// TIA Portal V15.1 export
// export: Created 2024-06-21T08:41:05.8674969Z, ExportSetting WithDefaults, DisplayName Totally Integrated Automation Portal, DisplayVersion V15.1 Update 5, DisplayName TIA Portal Openness, DisplayVersion V15.1 Update 5, DisplayName SINAMICS Startdrive Advanced, DisplayVersion V15.1, DisplayName G130, G150, S120, S150, SINAMICS MV, S210, DisplayVersion V15.1, DisplayName G110M, G120, G120C, G120D, G120P, DisplayVersion V15.1, DisplayName STEP 7 Professional, DisplayVersion V15.1 Update 5, DisplayName STEP 7 Safety, DisplayVersion V15.1, DisplayName WinCC Professional, DisplayVersion V15.1 Update 5, DisplayName SIMATIC Visualization Architect, DisplayVersion V15.1
FUNCTION_BLOCK "LGBDanfoss-FC302PN"   // FB6600, FBD
TITLE = LGBDanfoss-FC302PN
{ S7_Optimized_Access := 'TRUE' }
AUTHOR : VCC
FAMILY : Actuator
NAME : Danfoss
VERSION : 0.1
// ============================================================================  Block to control a frequency controller Danfoss FC302 on ProfiNET.  ============================================================================
// stored: AutoNumber false, IsIECCheckEnabled false, IsRetainMemResEnabled false, MemoryReserve 100, SetENOAutomatically False, UDAEnableTagReadback false
   VAR_INPUT
      I_ReferenceValueLSB { ExternalAccessible := 'False'; ExternalVisible := 'False'; ExternalWritable := 'False'} : Bool;   // Bit 0
      I_ReferenceValueMSB { ExternalAccessible := 'False'; ExternalVisible := 'False'; ExternalWritable := 'False'} : Bool;   // Bit 1
      I_DCBrake { ExternalAccessible := 'False'; ExternalVisible := 'False'; ExternalWritable := 'False'} : Bool;   // Bit 2
      I_Coasting { ExternalAccessible := 'False'; ExternalVisible := 'False'; ExternalWritable := 'False'} : Bool;   // Bit 3
      I_QuickStop { ExternalAccessible := 'False'; ExternalVisible := 'False'; ExternalWritable := 'False'} : Bool;   // Bit 4
      I_HoldOutputFreq { ExternalAccessible := 'False'; ExternalVisible := 'False'; ExternalWritable := 'False'} : Bool;   // Bit 5
      I_RampStopStart { ExternalAccessible := 'False'; ExternalVisible := 'False'; ExternalWritable := 'False'} : Bool;   // Bit 6
      I_Reset { ExternalAccessible := 'False'; ExternalVisible := 'False'; ExternalWritable := 'False'} : Bool;   // Bit 7
      I_Jog { ExternalAccessible := 'False'; ExternalVisible := 'False'; ExternalWritable := 'False'} : Bool;   // Bit 8
      I_RampSelection { ExternalAccessible := 'False'; ExternalVisible := 'False'; ExternalWritable := 'False'} : Bool;   // Bit 9
      I_DataValid { ExternalAccessible := 'False'; ExternalVisible := 'False'; ExternalWritable := 'False'} : Bool;   // Bit 10
      I_Relay01 { ExternalAccessible := 'False'; ExternalVisible := 'False'; ExternalWritable := 'False'} : Bool;   // Bit 11
      I_Relay04 { ExternalAccessible := 'False'; ExternalVisible := 'False'; ExternalWritable := 'False'} : Bool;   // Bit 12
      I_SetupSelectionLSB { ExternalAccessible := 'False'; ExternalVisible := 'False'; ExternalWritable := 'False'} : Bool;   // Bit 13
      I_SetupSelectionMSB { ExternalAccessible := 'False'; ExternalVisible := 'False'; ExternalWritable := 'False'} : Bool;   // Bit 14
      I_Reverse { ExternalAccessible := 'False'; ExternalVisible := 'False'; ExternalWritable := 'False'} : Bool;   // Bit 15
      C_HWSubInput { ExternalAccessible := 'False'; ExternalVisible := 'False'; ExternalWritable := 'False'} : HW_SUBMODULE;   // I/O
      C_HWSubOutput { ExternalAccessible := 'False'; ExternalVisible := 'False'; ExternalWritable := 'False'} : HW_SUBMODULE;   // I/O
      I_MRV_FC { ExternalAccessible := 'False'; ExternalVisible := 'False'; ExternalWritable := 'False'} : Real;   // Main Reference Value (0-4000Hex = 0 - 100 %)
      I_PCDIndex3 { ExternalAccessible := 'False'; ExternalVisible := 'False'; ExternalWritable := 'False'} : Int;   // Process data index 3
      I_PCDIndex4 { ExternalAccessible := 'False'; ExternalVisible := 'False'; ExternalWritable := 'False'} : Int;   // Process data index 4
      I_PCDIndex5 { ExternalAccessible := 'False'; ExternalVisible := 'False'; ExternalWritable := 'False'} : Int;   // Process data index 5
      I_PCDIndex6 { ExternalAccessible := 'False'; ExternalVisible := 'False'; ExternalWritable := 'False'} : Int;   // Process data index 6
      I_PCDIndex7 { ExternalAccessible := 'False'; ExternalVisible := 'False'; ExternalWritable := 'False'} : Int;   // Process data index 7
      I_PCDIndex8 { ExternalAccessible := 'False'; ExternalVisible := 'False'; ExternalWritable := 'False'} : Int;   // Process data index 8
      I_PCDIndex9 { ExternalAccessible := 'False'; ExternalVisible := 'False'; ExternalWritable := 'False'} : Int;   // Process data index 9
      I_PCDIndex10 { ExternalAccessible := 'False'; ExternalVisible := 'False'; ExternalWritable := 'False'} : Int;   // Process data index 10
   END_VAR
   VAR_OUTPUT
      O_FCReady { ExternalAccessible := 'False'; ExternalVisible := 'False'; ExternalWritable := 'False'} : Bool;
      O_DriveReady { ExternalAccessible := 'False'; ExternalVisible := 'False'; ExternalWritable := 'False'} : Bool;
      O_CoastingReady { ExternalAccessible := 'False'; ExternalVisible := 'False'; ExternalWritable := 'False'} : Bool;
      O_Trip { ExternalAccessible := 'False'; ExternalVisible := 'False'; ExternalWritable := 'False'} : Bool;
      O_Error { ExternalAccessible := 'False'; ExternalVisible := 'False'; ExternalWritable := 'False'} : Bool;
      O_NotUsed { ExternalAccessible := 'False'; ExternalVisible := 'False'; ExternalWritable := 'False'} : Bool;
      O_TripLock { ExternalAccessible := 'False'; ExternalVisible := 'False'; ExternalWritable := 'False'} : Bool;
      O_Warning { ExternalAccessible := 'False'; ExternalVisible := 'False'; ExternalWritable := 'False'} : Bool;
      O_SpeedOK { ExternalAccessible := 'False'; ExternalVisible := 'False'; ExternalWritable := 'False'} : Bool;
      O_BusControl { ExternalAccessible := 'False'; ExternalVisible := 'False'; ExternalWritable := 'False'} : Bool;
      O_FrequencyLimit { ExternalAccessible := 'False'; ExternalVisible := 'False'; ExternalWritable := 'False'} : Bool;
      O_InOperation { ExternalAccessible := 'False'; ExternalVisible := 'False'; ExternalWritable := 'False'} : Bool;
      O_Autostart { ExternalAccessible := 'False'; ExternalVisible := 'False'; ExternalWritable := 'False'} : Bool;
      O_VoltageLimExceed { ExternalAccessible := 'False'; ExternalVisible := 'False'; ExternalWritable := 'False'} : Bool;
      O_TorqueLimExceed { ExternalAccessible := 'False'; ExternalVisible := 'False'; ExternalWritable := 'False'} : Bool;
      O_TimerLimExceed { ExternalAccessible := 'False'; ExternalVisible := 'False'; ExternalWritable := 'False'} : Bool;
      O_ActualSpeed { ExternalAccessible := 'False'; ExternalVisible := 'False'; ExternalWritable := 'False'} : Real;
      H_FromFC_STW { ExternalAccessible := 'False'; ExternalVisible := 'False'; ExternalWritable := 'False'} : Word;
      H_FromFC_MAV { ExternalAccessible := 'False'; ExternalVisible := 'False'; ExternalWritable := 'False'} : Int;
      H_MAV_Procent { ExternalAccessible := 'False'; ExternalVisible := 'False'; ExternalWritable := 'False'} : Int;
      H_FromFC_Warning { ExternalAccessible := 'False'; ExternalVisible := 'False'; ExternalWritable := 'False'} : DWord;
      H_FromFC_Alarm { ExternalAccessible := 'False'; ExternalVisible := 'False'; ExternalWritable := 'False'} : DWord;
      H_FromFC_MotorCurrent { ExternalAccessible := 'False'; ExternalVisible := 'False'; ExternalWritable := 'False'} : Int;
      H_FromFC_MotorTorque { ExternalAccessible := 'False'; ExternalVisible := 'False'; ExternalWritable := 'False'} : Int;
      H_FromFC_MotorFrequency { ExternalAccessible := 'False'; ExternalVisible := 'False'; ExternalWritable := 'False'} : Int;
      H_FromFC_Spare { ExternalAccessible := 'False'; ExternalVisible := 'False'; ExternalWritable := 'False'} : Word;
      H_ToFC_CTW { ExternalAccessible := 'False'; ExternalVisible := 'False'; ExternalWritable := 'False'} : Word;
      H_MRV_Procent { ExternalAccessible := 'False'; ExternalVisible := 'False'; ExternalWritable := 'False'} : Real;
      H_ToFC_MRV { ExternalAccessible := 'False'; ExternalVisible := 'False'; ExternalWritable := 'False'} : Int;
   END_VAR
   VAR
      RampStopStart { ExternalAccessible := 'False'; ExternalVisible := 'False'; ExternalWritable := 'False'} : Bool;
      HvEdgeRampStopStart { ExternalAccessible := 'False'; ExternalVisible := 'False'; ExternalWritable := 'False'} : Bool;
      RetValueDataFromFC { ExternalAccessible := 'False'; ExternalVisible := 'False'; ExternalWritable := 'False'} : Int;
      RetValueDataToFC { ExternalAccessible := 'False'; ExternalVisible := 'False'; ExternalWritable := 'False'} : Int;
      ActualSpeed { ExternalAccessible := 'False'; ExternalVisible := 'False'; ExternalWritable := 'False'} : Real;
      InDataDrive { ExternalAccessible := 'False'; ExternalVisible := 'False'; ExternalWritable := 'False'} : Array[1..10] of Word;   // Data from Drive
      Read { ExternalAccessible := 'False'; ExternalVisible := 'False'; ExternalWritable := 'False'} : Struct
         STW { ExternalAccessible := 'False'; ExternalVisible := 'False'; ExternalWritable := 'False'} : Struct
            SpeedOK { ExternalAccessible := 'False'; ExternalVisible := 'False'; ExternalWritable := 'False'} : Bool;
            BusControl { ExternalAccessible := 'False'; ExternalVisible := 'False'; ExternalWritable := 'False'} : Bool;
            FrequencyLimit { ExternalAccessible := 'False'; ExternalVisible := 'False'; ExternalWritable := 'False'} : Bool;
            InOperation { ExternalAccessible := 'False'; ExternalVisible := 'False'; ExternalWritable := 'False'} : Bool;
            Autostart { ExternalAccessible := 'False'; ExternalVisible := 'False'; ExternalWritable := 'False'} : Bool;
            VoltageLimitExceed { ExternalAccessible := 'False'; ExternalVisible := 'False'; ExternalWritable := 'False'} : Bool;
            TorqueLimitExceed { ExternalAccessible := 'False'; ExternalVisible := 'False'; ExternalWritable := 'False'} : Bool;
            TimerLimitExceed { ExternalAccessible := 'False'; ExternalVisible := 'False'; ExternalWritable := 'False'} : Bool;
            ControlReady { ExternalAccessible := 'False'; ExternalVisible := 'False'; ExternalWritable := 'False'} : Bool;
            DriveReady { ExternalAccessible := 'False'; ExternalVisible := 'False'; ExternalWritable := 'False'} : Bool;
            CostingStop { ExternalAccessible := 'False'; ExternalVisible := 'False'; ExternalWritable := 'False'} : Bool;
            Trip { ExternalAccessible := 'False'; ExternalVisible := 'False'; ExternalWritable := 'False'} : Bool;
            Error { ExternalAccessible := 'False'; ExternalVisible := 'False'; ExternalWritable := 'False'} : Bool;
            NotUsed { ExternalAccessible := 'False'; ExternalVisible := 'False'; ExternalWritable := 'False'} : Bool;
            TripLock { ExternalAccessible := 'False'; ExternalVisible := 'False'; ExternalWritable := 'False'} : Bool;
            Warning { ExternalAccessible := 'False'; ExternalVisible := 'False'; ExternalWritable := 'False'} : Bool;
         END_STRUCT;
         MAV { ExternalAccessible := 'False'; ExternalVisible := 'False'; ExternalWritable := 'False'} : Int;
         WarningStatus { ExternalAccessible := 'False'; ExternalVisible := 'False'; ExternalWritable := 'False'} : DWord;   // Hex
         AlarmStatus { ExternalAccessible := 'False'; ExternalVisible := 'False'; ExternalWritable := 'False'} : DWord;   // Hex
         MotorCurrent { ExternalAccessible := 'False'; ExternalVisible := 'False'; ExternalWritable := 'False'} : Int;   // Motor current (xx.xx A)
         MotorTorque { ExternalAccessible := 'False'; ExternalVisible := 'False'; ExternalWritable := 'False'} : Int;   // Torque (%)
         MotorFrequencey { ExternalAccessible := 'False'; ExternalVisible := 'False'; ExternalWritable := 'False'} : Int;
         PCDSpare { ExternalAccessible := 'False'; ExternalVisible := 'False'; ExternalWritable := 'False'} : Word;
      END_STRUCT;
      Write { ExternalAccessible := 'False'; ExternalVisible := 'False'; ExternalWritable := 'False'} : Struct
         CTW { ExternalAccessible := 'False'; ExternalVisible := 'False'; ExternalWritable := 'False'} : Struct
            Jog { ExternalAccessible := 'False'; ExternalVisible := 'False'; ExternalWritable := 'False'} : Bool;
            RampSelection { ExternalAccessible := 'False'; ExternalVisible := 'False'; ExternalWritable := 'False'} : Bool;
            DataValid { ExternalAccessible := 'False'; ExternalVisible := 'False'; ExternalWritable := 'False'} : Bool;
            Relay01 { ExternalAccessible := 'False'; ExternalVisible := 'False'; ExternalWritable := 'False'} : Bool;
            Relay02 { ExternalAccessible := 'False'; ExternalVisible := 'False'; ExternalWritable := 'False'} : Bool;
            SetupSelectionLSB { ExternalAccessible := 'False'; ExternalVisible := 'False'; ExternalWritable := 'False'} : Bool;
            SetupSelectionMSB { ExternalAccessible := 'False'; ExternalVisible := 'False'; ExternalWritable := 'False'} : Bool;
            Reverse { ExternalAccessible := 'False'; ExternalVisible := 'False'; ExternalWritable := 'False'} : Bool;
            ReferenceValueLSB { ExternalAccessible := 'False'; ExternalVisible := 'False'; ExternalWritable := 'False'} : Bool;
            ReferenceValueMSB { ExternalAccessible := 'False'; ExternalVisible := 'False'; ExternalWritable := 'False'} : Bool;
            DCBrake { ExternalAccessible := 'False'; ExternalVisible := 'False'; ExternalWritable := 'False'} : Bool;
            Coasting { ExternalAccessible := 'False'; ExternalVisible := 'False'; ExternalWritable := 'False'} : Bool;
            QuickStop { ExternalAccessible := 'False'; ExternalVisible := 'False'; ExternalWritable := 'False'} : Bool;
            HoldOutputFreq { ExternalAccessible := 'False'; ExternalVisible := 'False'; ExternalWritable := 'False'} : Bool;
            RampStopStart { ExternalAccessible := 'False'; ExternalVisible := 'False'; ExternalWritable := 'False'} : Bool;
            Reset { ExternalAccessible := 'False'; ExternalVisible := 'False'; ExternalWritable := 'False'} : Bool;
         END_STRUCT;
         MRV { ExternalAccessible := 'False'; ExternalVisible := 'False'; ExternalWritable := 'False'} : Int;
         PCDSpare { ExternalAccessible := 'False'; ExternalVisible := 'False'; ExternalWritable := 'False'} : Array[3..10] of Word;
      END_STRUCT;
   END_VAR
   VAR_TEMP   // added for the SCL form of the ladder/FBD networks
      _w1 : Bool;
   END_VAR
BEGIN

REGION Network 1: **** 1 - Inputs **** Communication drive
   // Communication with drive
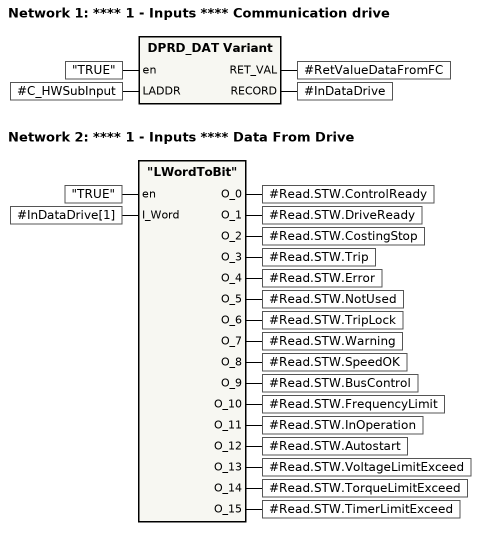
   IF "TRUE" THEN #RetValueDataFromFC := DPRD_DAT(LADDR := #C_HWSubInput, RECORD => #InDataDrive); END_IF;
END_REGION

REGION Network 2: **** 1 - Inputs **** Data From Drive
   // Data From Drive
   IF "TRUE" THEN
       "LWordToBit"(I_Word := #InDataDrive[1],
                    O_0 => #Read.STW.ControlReady,
                    O_1 => #Read.STW.DriveReady,
                    O_2 => #Read.STW.CostingStop,
                    O_3 => #Read.STW.Trip,
                    O_4 => #Read.STW.Error,
                    O_5 => #Read.STW.NotUsed,
                    O_6 => #Read.STW.TripLock,
                    O_7 => #Read.STW.Warning,
                    O_8 => #Read.STW.SpeedOK,
                    O_9 => #Read.STW.BusControl,
                    O_10 => #Read.STW.FrequencyLimit,
                    O_11 => #Read.STW.InOperation,
                    O_12 => #Read.STW.Autostart,
                    O_13 => #Read.STW.VoltageLimitExceed,
                    O_14 => #Read.STW.TorqueLimitExceed,
                    O_15 => #Read.STW.TimerLimitExceed);
   END_IF;
END_REGION

REGION Network 3: **** 1 - Inputs **** Data From Drive
   // Data From Drive
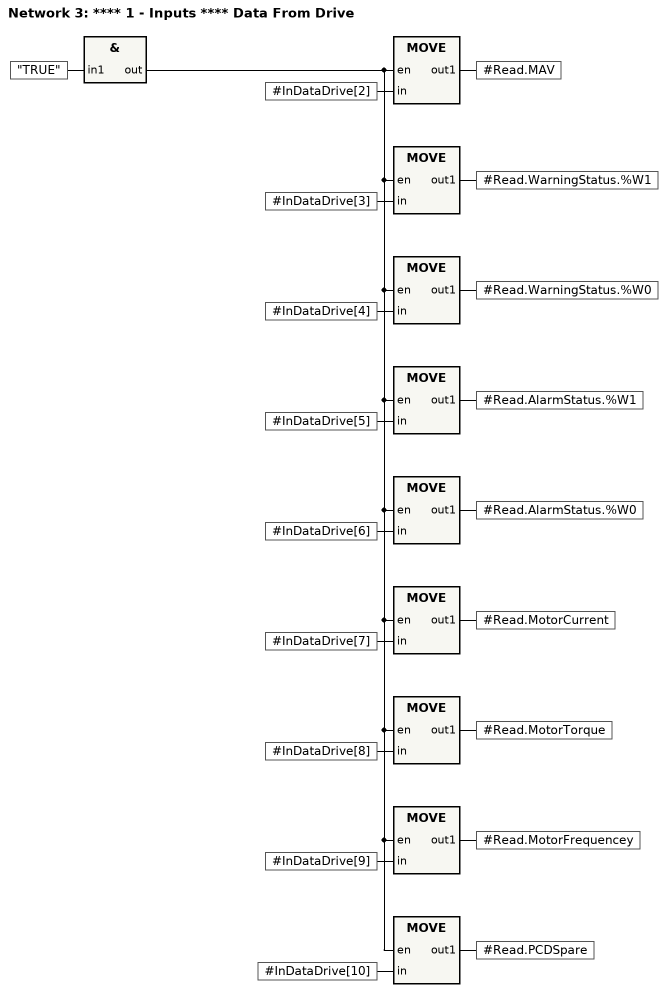
   IF "TRUE" THEN
       #Read.MAV := #InDataDrive[2];
       #Read.WarningStatus.%W1 := #InDataDrive[3];
       #Read.WarningStatus.%W0 := #InDataDrive[4];
       #Read.AlarmStatus.%W1 := #InDataDrive[5];
       #Read.AlarmStatus.%W0 := #InDataDrive[6];
       #Read.MotorCurrent := #InDataDrive[7];
       #Read.MotorTorque := #InDataDrive[8];
       #Read.MotorFrequencey := #InDataDrive[9];
       #Read.PCDSpare := #InDataDrive[10];
   END_IF;
END_REGION

REGION Network 4: **** 8 - Outputs **** STW
   // Frequency controller : STW (Status word)
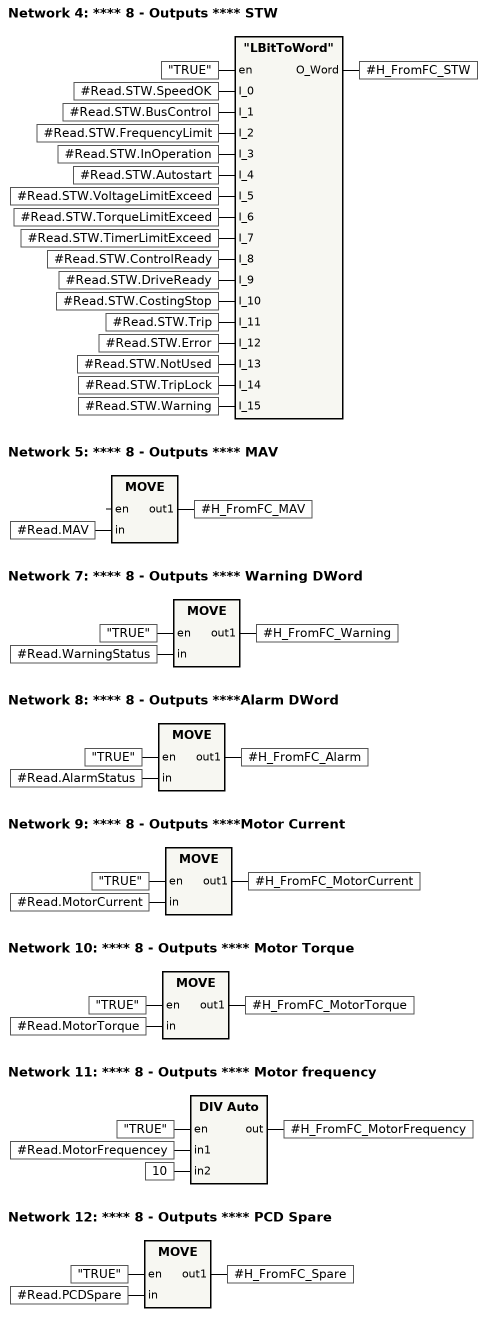
   IF "TRUE" THEN
       "LBitToWord"(I_0 := #Read.STW.SpeedOK,
                    I_1 := #Read.STW.BusControl,
                    I_2 := #Read.STW.FrequencyLimit,
                    I_3 := #Read.STW.InOperation,
                    I_4 := #Read.STW.Autostart,
                    I_5 := #Read.STW.VoltageLimitExceed,
                    I_6 := #Read.STW.TorqueLimitExceed,
                    I_7 := #Read.STW.TimerLimitExceed,
                    I_8 := #Read.STW.ControlReady,
                    I_9 := #Read.STW.DriveReady,
                    I_10 := #Read.STW.CostingStop,
                    I_11 := #Read.STW.Trip,
                    I_12 := #Read.STW.Error,
                    I_13 := #Read.STW.NotUsed,
                    I_14 := #Read.STW.TripLock,
                    I_15 := #Read.STW.Warning,
                    O_Word => #H_FromFC_STW);
   END_IF;
END_REGION

REGION Network 5: **** 8 - Outputs **** MAV
   // Frequency controller : MAV (Main reference Value - real value)
   #H_FromFC_MAV := #Read.MAV;
END_REGION

NETWORK
TITLE = **** 4.6 - Machine Status - Calculated **** Actual Speed
// Speed to MFP
      L     #Read.MAV;
      ITD;
      L     DINT#1000;
      *D;
      L     DW#16#4000;
      /D;
      T     #H_MAV_Procent;

      L     #H_MAV_Procent;
      ITD;
      DTR;
      L     10.0;
      /R;
      T     #ActualSpeed;

REGION Network 7: **** 8 - Outputs **** Warning DWord
   // Frequency controller : Warning DWord
   IF "TRUE" THEN #H_FromFC_Warning := #Read.WarningStatus; END_IF;
END_REGION

REGION Network 8: **** 8 - Outputs ****Alarm DWord
   // Frequency controller : Alarm DWord
   IF "TRUE" THEN #H_FromFC_Alarm := #Read.AlarmStatus; END_IF;
END_REGION

REGION Network 9: **** 8 - Outputs ****Motor Current
   // Frequency controller : Motor Current
   IF "TRUE" THEN #H_FromFC_MotorCurrent := #Read.MotorCurrent; END_IF;
END_REGION

REGION Network 10: **** 8 - Outputs **** Motor Torque
   // Frequency controller :  Motor Torque
   IF "TRUE" THEN #H_FromFC_MotorTorque := #Read.MotorTorque; END_IF;
END_REGION

REGION Network 11: **** 8 - Outputs **** Motor frequency
   // Frequency controller : Motor frequency
   IF "TRUE" THEN #H_FromFC_MotorFrequency := #Read.MotorFrequencey / 10; END_IF;
END_REGION

REGION Network 12: **** 8 - Outputs **** PCD Spare
   // Frequency controller : PCD Spare
   IF "TRUE" THEN #H_FromFC_Spare := #Read.PCDSpare; END_IF;
END_REGION

REGION Network 13: **** 8 - Outputs **** Reference LSB
   // CTW : Reference Value LSB
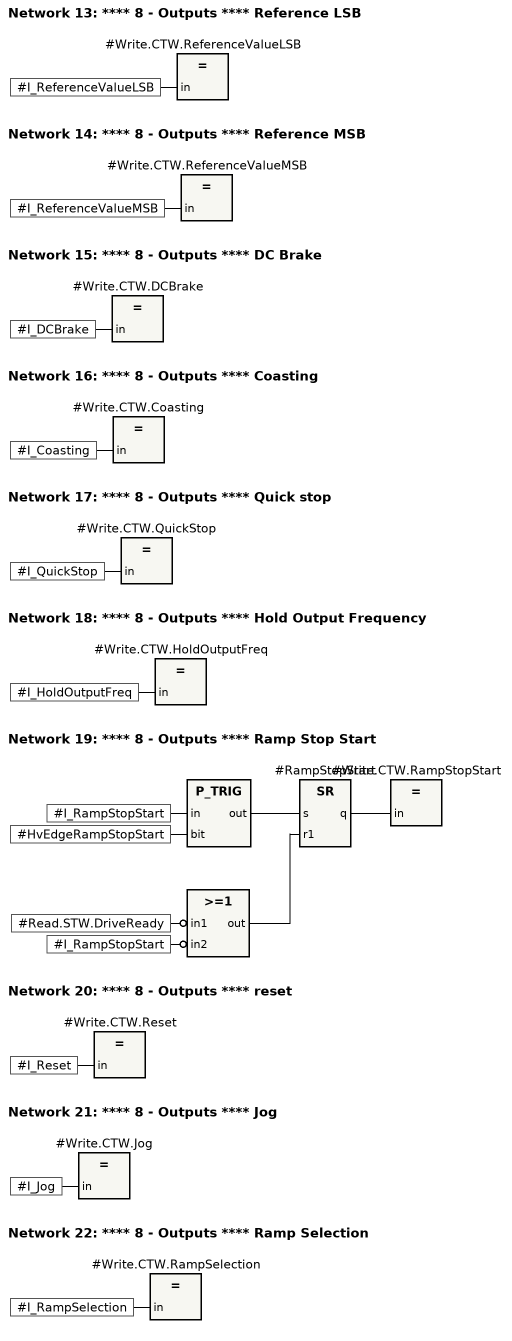
   #Write.CTW.ReferenceValueLSB := #I_ReferenceValueLSB;
END_REGION

REGION Network 14: **** 8 - Outputs **** Reference MSB
   // CTW : Reference Value MSB
   #Write.CTW.ReferenceValueMSB := #I_ReferenceValueMSB;
END_REGION

REGION Network 15: **** 8 - Outputs **** DC Brake
   // CTW : Index valid
   #Write.CTW.DCBrake := #I_DCBrake;
END_REGION

REGION Network 16: **** 8 - Outputs **** Coasting
   // CTW : Coasting
   #Write.CTW.Coasting := #I_Coasting;
END_REGION

REGION Network 17: **** 8 - Outputs **** Quick stop
   // CTW : Quick stop
   #Write.CTW.QuickStop := #I_QuickStop;
END_REGION

REGION Network 18: **** 8 - Outputs **** Hold Output Frequency
   // CTW : Hold Output Frequency
   #Write.CTW.HoldOutputFreq := #I_HoldOutputFreq;
END_REGION

REGION Network 19: **** 8 - Outputs **** Ramp Stop Start
   // CTW : Reverse
   #_w1 := #I_RampStopStart AND NOT #HvEdgeRampStopStart;   // rising edge
   #HvEdgeRampStopStart := #I_RampStopStart;
   IF #_w1 THEN
       #RampStopStart := TRUE;   // SR flip-flop
   END_IF;
   IF NOT #Read.STW.DriveReady OR NOT #I_RampStopStart THEN #RampStopStart := FALSE; END_IF;
   #Write.CTW.RampStopStart := #RampStopStart;
END_REGION

REGION Network 20: **** 8 - Outputs **** reset
   // CTW : reset
   #Write.CTW.Reset := #I_Reset;
END_REGION

REGION Network 21: **** 8 - Outputs **** Jog
   // CTW : Jog
   #Write.CTW.Jog := #I_Jog;
END_REGION

REGION Network 22: **** 8 - Outputs **** Ramp Selection
   // CTW : Ramp Selection
   #Write.CTW.RampSelection := #I_RampSelection;
END_REGION

REGION Network 23: **** 8 - Outputs **** DataValid
   // CTW : DataValid
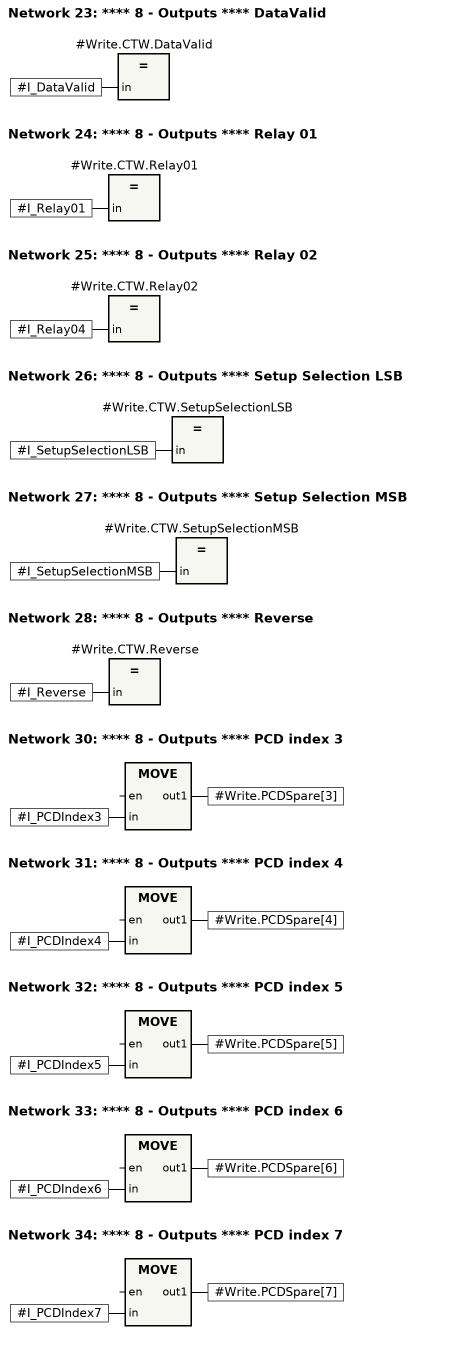
   #Write.CTW.DataValid := #I_DataValid;
END_REGION

REGION Network 24: **** 8 - Outputs **** Relay 01
   // CTW : Relay 01
   #Write.CTW.Relay01 := #I_Relay01;
END_REGION

REGION Network 25: **** 8 - Outputs **** Relay 02
   // CTW : Relay 04
   #Write.CTW.Relay02 := #I_Relay04;
END_REGION

REGION Network 26: **** 8 - Outputs **** Setup Selection LSB
   // CTW : #Setup Selection LSB
   #Write.CTW.SetupSelectionLSB := #I_SetupSelectionLSB;
END_REGION

REGION Network 27: **** 8 - Outputs **** Setup Selection MSB
   // CTW : #Setup Selection MSB
   #Write.CTW.SetupSelectionMSB := #I_SetupSelectionMSB;
END_REGION

REGION Network 28: **** 8 - Outputs **** Reverse
   // CTW : Reverse
   #Write.CTW.Reverse := #I_Reverse;
END_REGION

NETWORK
TITLE = **** 4.6 - Machine Status - Calculated **** Setpoint Speed
// Speed to MFP
      L     #I_MRV_FC;
      L     16384.0;
      *R;
      L     100.0;
      /R;
      RND;
      T     #Write.MRV;

REGION Network 30: **** 8 - Outputs **** PCD index 3
   // Selection of PCD index 3
   #Write.PCDSpare[3] := #I_PCDIndex3;
END_REGION

REGION Network 31: **** 8 - Outputs **** PCD index 4
   // Selection of PCD index 4
   #Write.PCDSpare[4] := #I_PCDIndex4;
END_REGION

REGION Network 32: **** 8 - Outputs **** PCD index 5
   // Selection of PCD index 5
   #Write.PCDSpare[5] := #I_PCDIndex5;
END_REGION

REGION Network 33: **** 8 - Outputs **** PCD index 6
   // Selection of PCD index 6
   #Write.PCDSpare[6] := #I_PCDIndex6;
END_REGION

REGION Network 34: **** 8 - Outputs **** PCD index 7
   // Selection of PCD index 7
   #Write.PCDSpare[7] := #I_PCDIndex7;
END_REGION

REGION Network 35: **** 8 - Outputs **** PCD index 8
   // Selection of PCD index 8
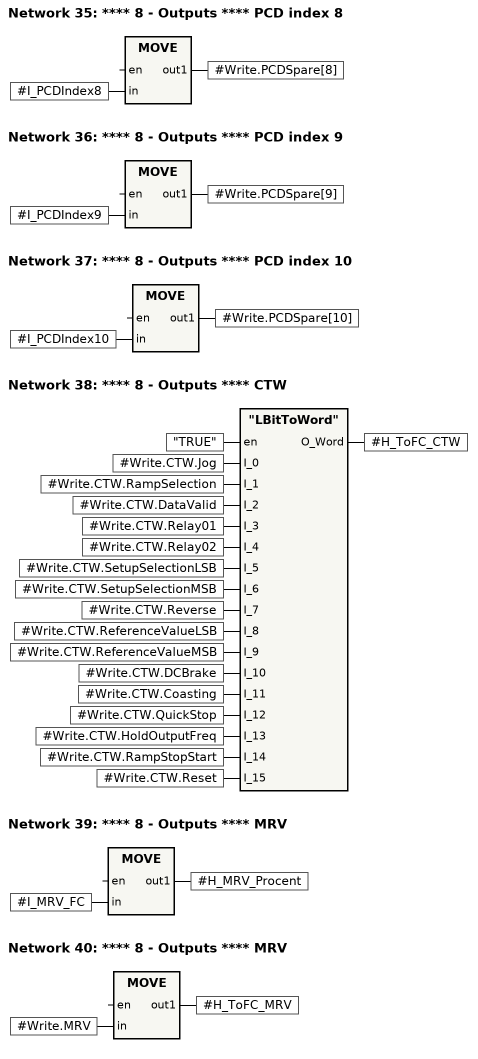
   #Write.PCDSpare[8] := #I_PCDIndex8;
END_REGION

REGION Network 36: **** 8 - Outputs **** PCD index 9
   // Selection of PCD index 9
   #Write.PCDSpare[9] := #I_PCDIndex9;
END_REGION

REGION Network 37: **** 8 - Outputs **** PCD index 10
   // Selection of PCD index 10
   #Write.PCDSpare[10] := #I_PCDIndex10;
END_REGION

REGION Network 38: **** 8 - Outputs **** CTW
   // Frequency controller : CTW (Control word)
   IF "TRUE" THEN
       "LBitToWord"(I_0 := #Write.CTW.Jog,
                    I_1 := #Write.CTW.RampSelection,
                    I_2 := #Write.CTW.DataValid,
                    I_3 := #Write.CTW.Relay01,
                    I_4 := #Write.CTW.Relay02,
                    I_5 := #Write.CTW.SetupSelectionLSB,
                    I_6 := #Write.CTW.SetupSelectionMSB,
                    I_7 := #Write.CTW.Reverse,
                    I_8 := #Write.CTW.ReferenceValueLSB,
                    I_9 := #Write.CTW.ReferenceValueMSB,
                    I_10 := #Write.CTW.DCBrake,
                    I_11 := #Write.CTW.Coasting,
                    I_12 := #Write.CTW.QuickStop,
                    I_13 := #Write.CTW.HoldOutputFreq,
                    I_14 := #Write.CTW.RampStopStart,
                    I_15 := #Write.CTW.Reset,
                    O_Word => #H_ToFC_CTW);
   END_IF;
END_REGION

REGION Network 39: **** 8 - Outputs **** MRV
   // Frequency controller : MRV (Main reference Value)
   #H_MRV_Procent := #I_MRV_FC;
END_REGION

REGION Network 40: **** 8 - Outputs **** MRV
   // Frequency controller : MRV (Main reference Value)
   #H_ToFC_MRV := #Write.MRV;
END_REGION

REGION Network 41: **** 8 - Outputs ****
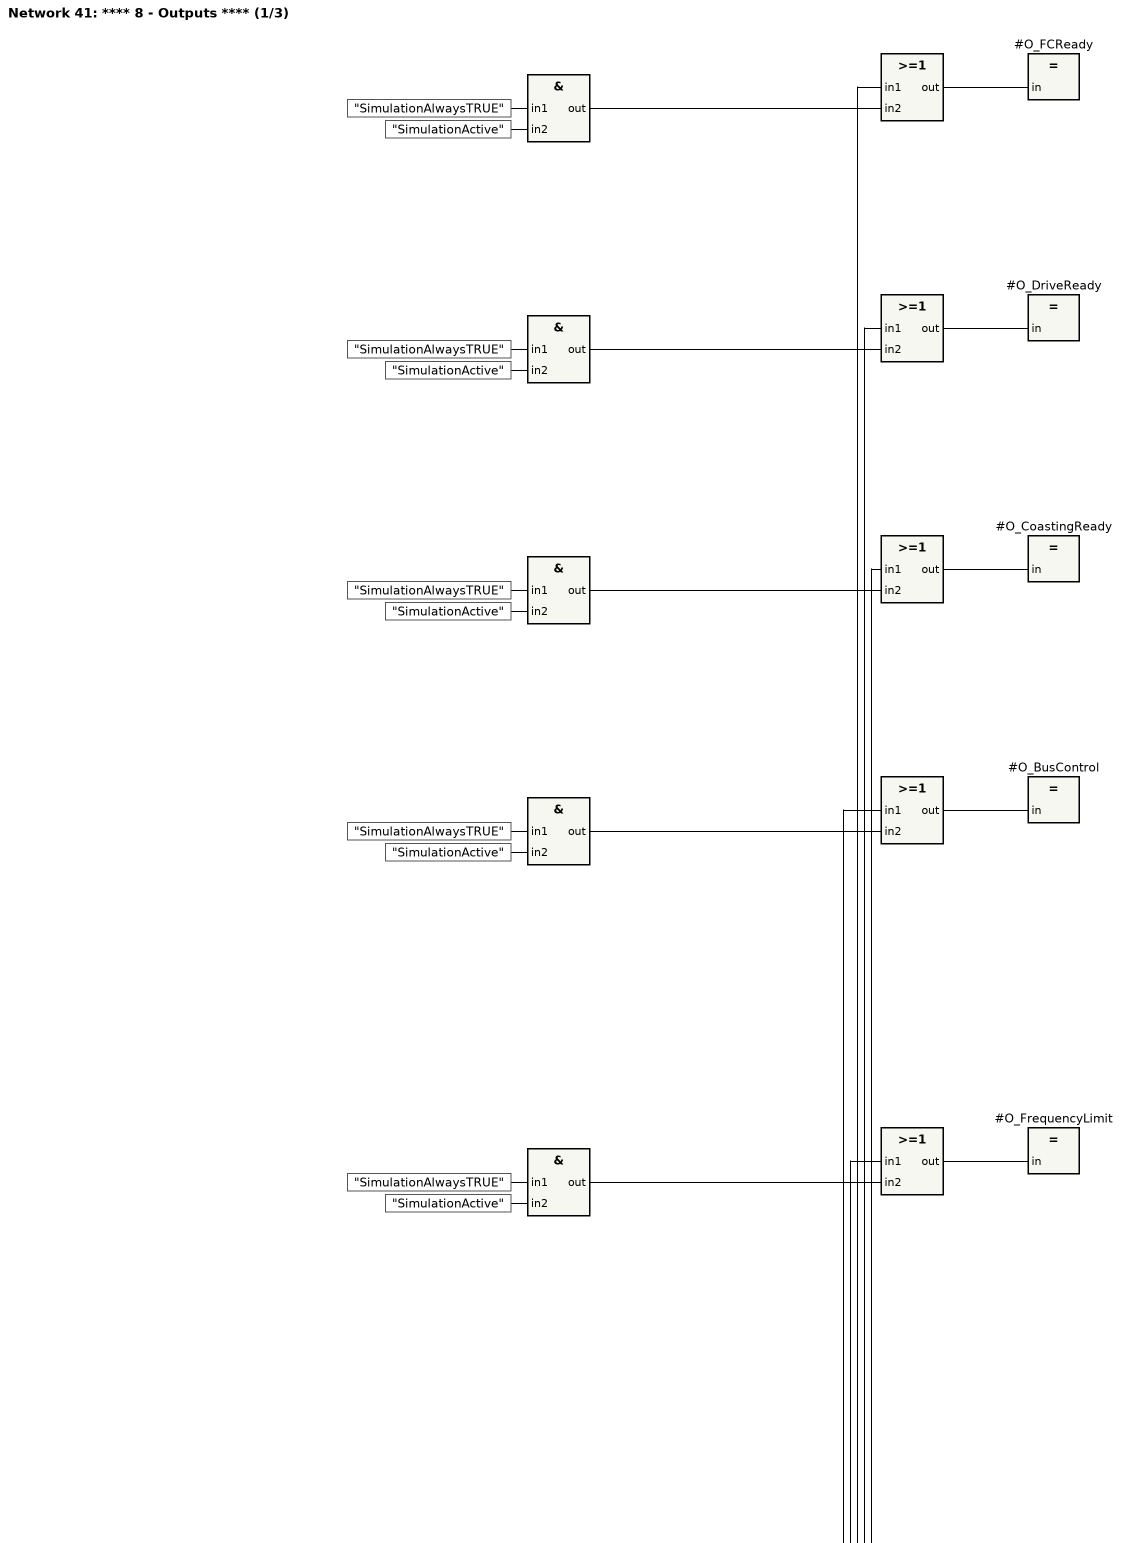
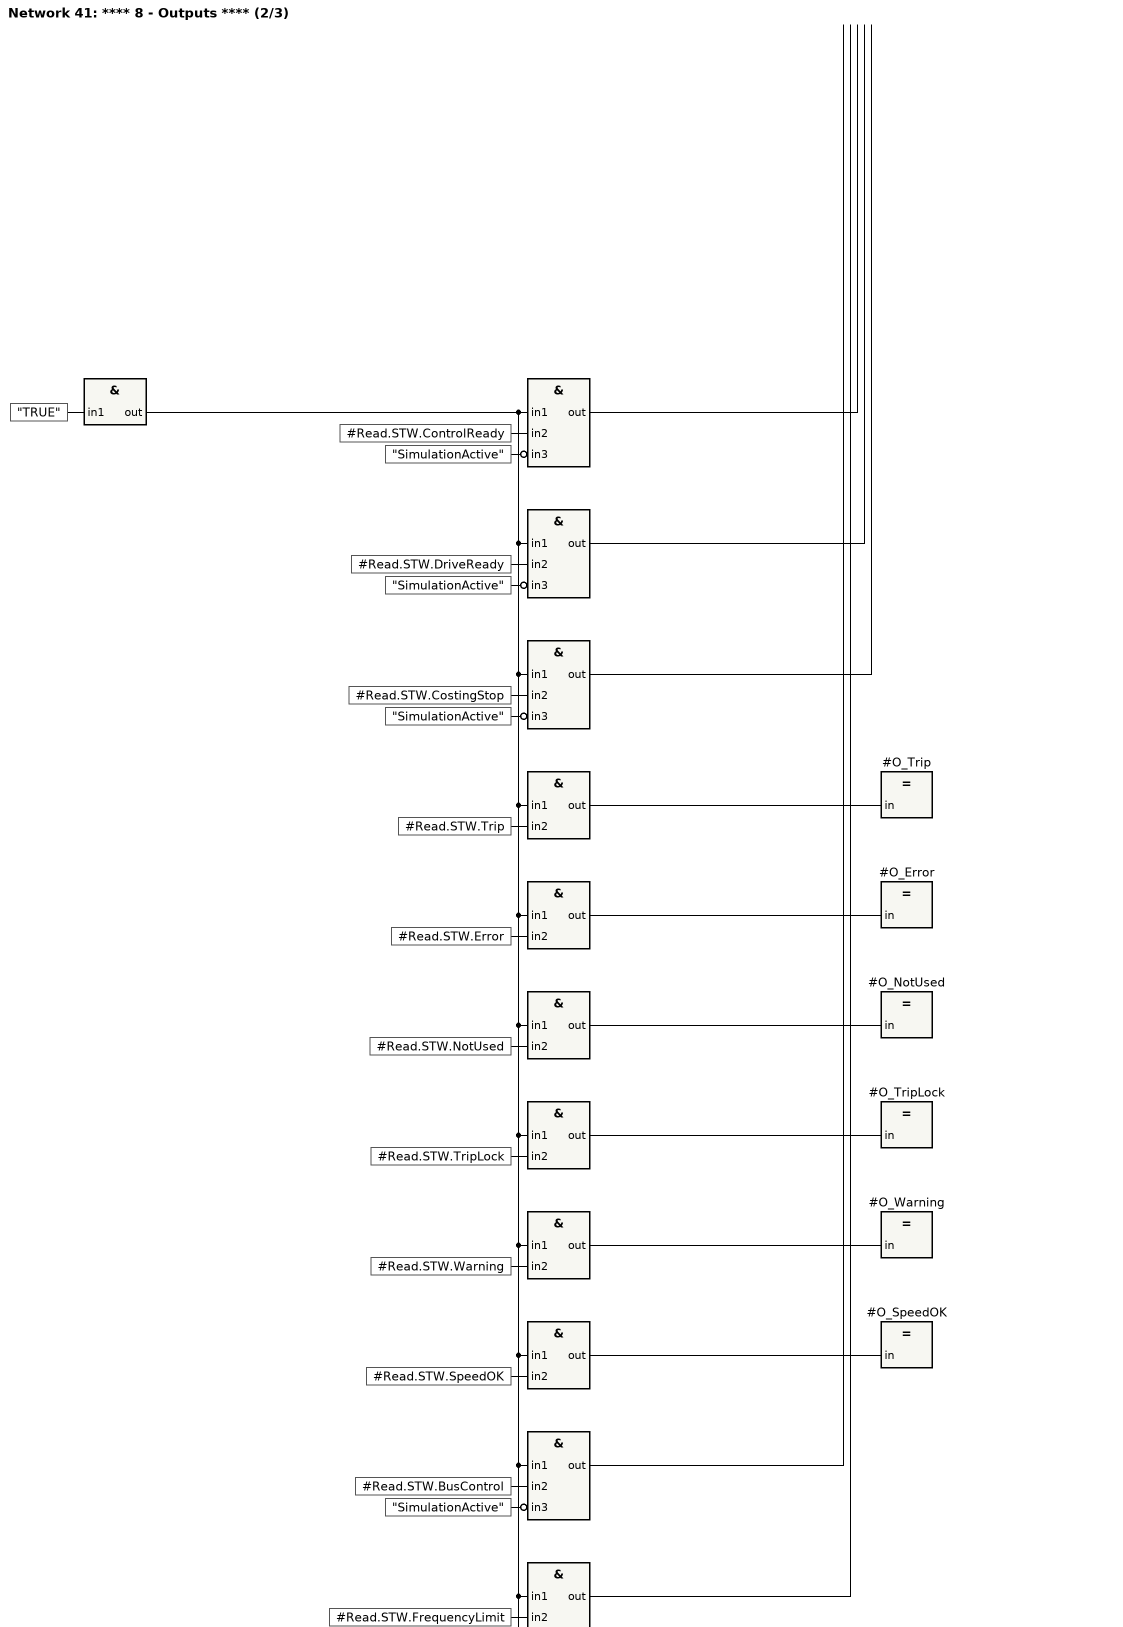
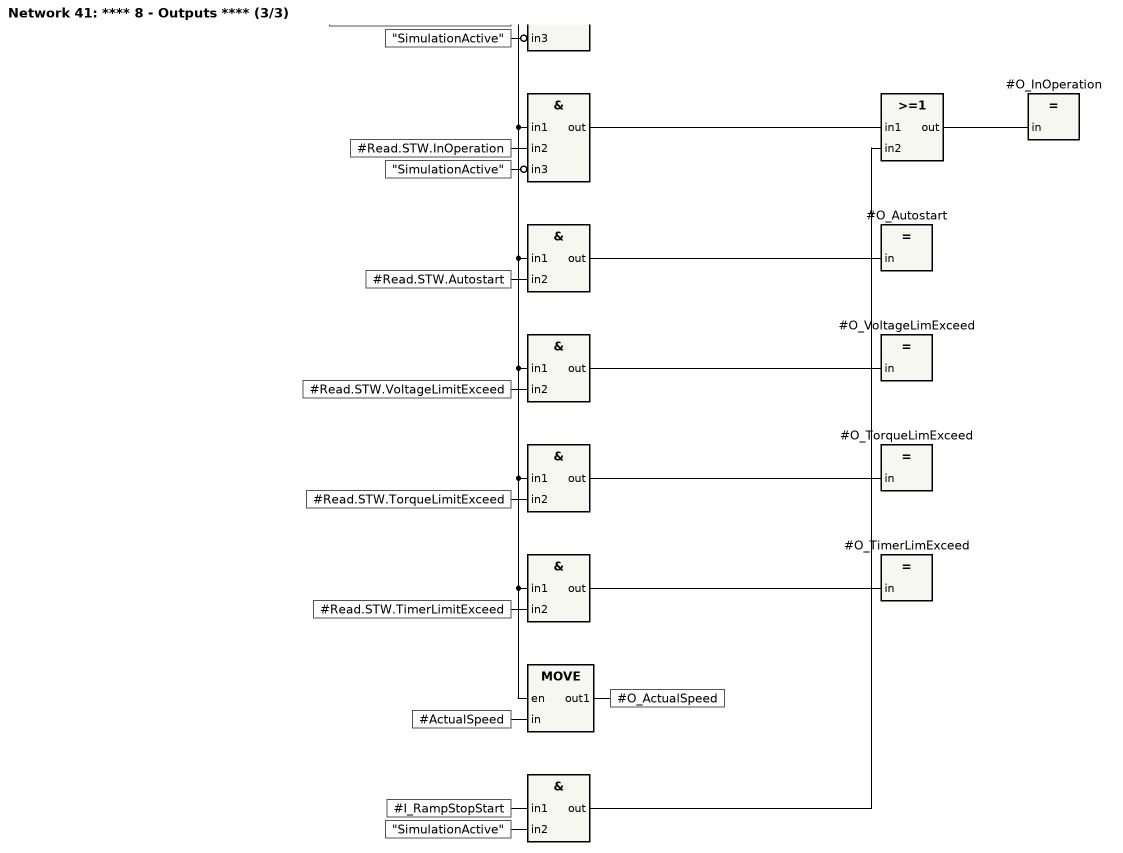
   #O_FCReady := ("TRUE" AND #Read.STW.ControlReady AND NOT "SimulationActive") OR ("SimulationAlwaysTRUE" AND "SimulationActive");
   #O_DriveReady := ("TRUE" AND #Read.STW.DriveReady AND NOT "SimulationActive") OR ("SimulationAlwaysTRUE" AND "SimulationActive");
   #O_CoastingReady := ("TRUE" AND #Read.STW.CostingStop AND NOT "SimulationActive") OR ("SimulationAlwaysTRUE" AND "SimulationActive");
   #O_Trip := "TRUE" AND #Read.STW.Trip;
   #O_Error := "TRUE" AND #Read.STW.Error;
   #O_NotUsed := "TRUE" AND #Read.STW.NotUsed;
   #O_TripLock := "TRUE" AND #Read.STW.TripLock;
   #O_Warning := "TRUE" AND #Read.STW.Warning;
   #O_SpeedOK := "TRUE" AND #Read.STW.SpeedOK;
   #O_BusControl := ("TRUE" AND #Read.STW.BusControl AND NOT "SimulationActive") OR ("SimulationAlwaysTRUE" AND "SimulationActive");
   #O_FrequencyLimit := ("TRUE" AND #Read.STW.FrequencyLimit AND NOT "SimulationActive") OR ("SimulationAlwaysTRUE" AND "SimulationActive");
   #O_InOperation := ("TRUE" AND #Read.STW.InOperation AND NOT "SimulationActive") OR (#I_RampStopStart AND "SimulationActive");
   #O_Autostart := "TRUE" AND #Read.STW.Autostart;
   #O_VoltageLimExceed := "TRUE" AND #Read.STW.VoltageLimitExceed;
   #O_TorqueLimExceed := "TRUE" AND #Read.STW.TorqueLimitExceed;
   #O_TimerLimExceed := "TRUE" AND #Read.STW.TimerLimitExceed;
   IF "TRUE" THEN #O_ActualSpeed := #ActualSpeed; END_IF;
END_REGION

REGION Network 42: **** 8 - Outputs **** data to Frequency controller
   // Write consistant data to Frequency controller
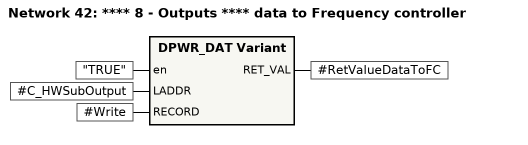
   IF "TRUE" THEN #RetValueDataToFC := DPWR_DAT(LADDR := #C_HWSubOutput, RECORD := #Write); END_IF;
END_REGION
END_FUNCTION_BLOCK
